(* PLC project Sin nombre, Desconocido Sin nombre 1 *)
(* stored: creationDateTime 2024-10-27T00:44:48, modificationDateTime 2024-10-28T16:29:27 *)

PROGRAM program0
  VAR
    timer : BOOL := 1;
    probar_sig : BOOL := 0;
    entro : BOOL := 0;
    entro0 : BOOL := 0;
    timer_corrido : BOOL := 0;
    acumular : BOOL := 0;
    hubo_cambio : BOOL := 0;  (* 0 *)
    luz1 : BOOL := 0;  (* darle ubic *)
    luz2 : BOOL := 0;  (* darle ubic *)
  END_VAR
  VAR
    sensor AT %IW0.0 : UINT := 34500;
  END_VAR
  VAR
    acum : UINT := 60000;
    tope_normal : UINT := 60;
    tope_alto : UINT := 40000;
    tope_superior : UINT := 0;
    actual : INT := 3;
    TON2 : TON;
    TP0 : TP;
    TOF1 : TOF;
    TP3 : TP;
    TON1 : TON;
    TON4 : TON;
    TON3 : TON;
    TON0 : TON;
    TON6 : TON;
  END_VAR
  VAR  (* added by the conversion: wires and edge detectors of the diagram *)
    _ADD78_ENO : BOOL;
    _ADD78_OUT : UINT;
    _EQ5_ENO : BOOL;
    _EQ5_OUT : BOOL;
    _GE83_ENO : BOOL;
    _GE83_OUT : BOOL;
    _ADD16_ENO : BOOL;
    _ADD16_OUT : INT;
    _EQ32_ENO : BOOL;
    _EQ32_OUT : BOOL;
    _GE55_ENO : BOOL;
    _GE55_OUT : BOOL;
    _LT97_ENO : BOOL;
    _LT97_OUT : BOOL;
  END_VAR

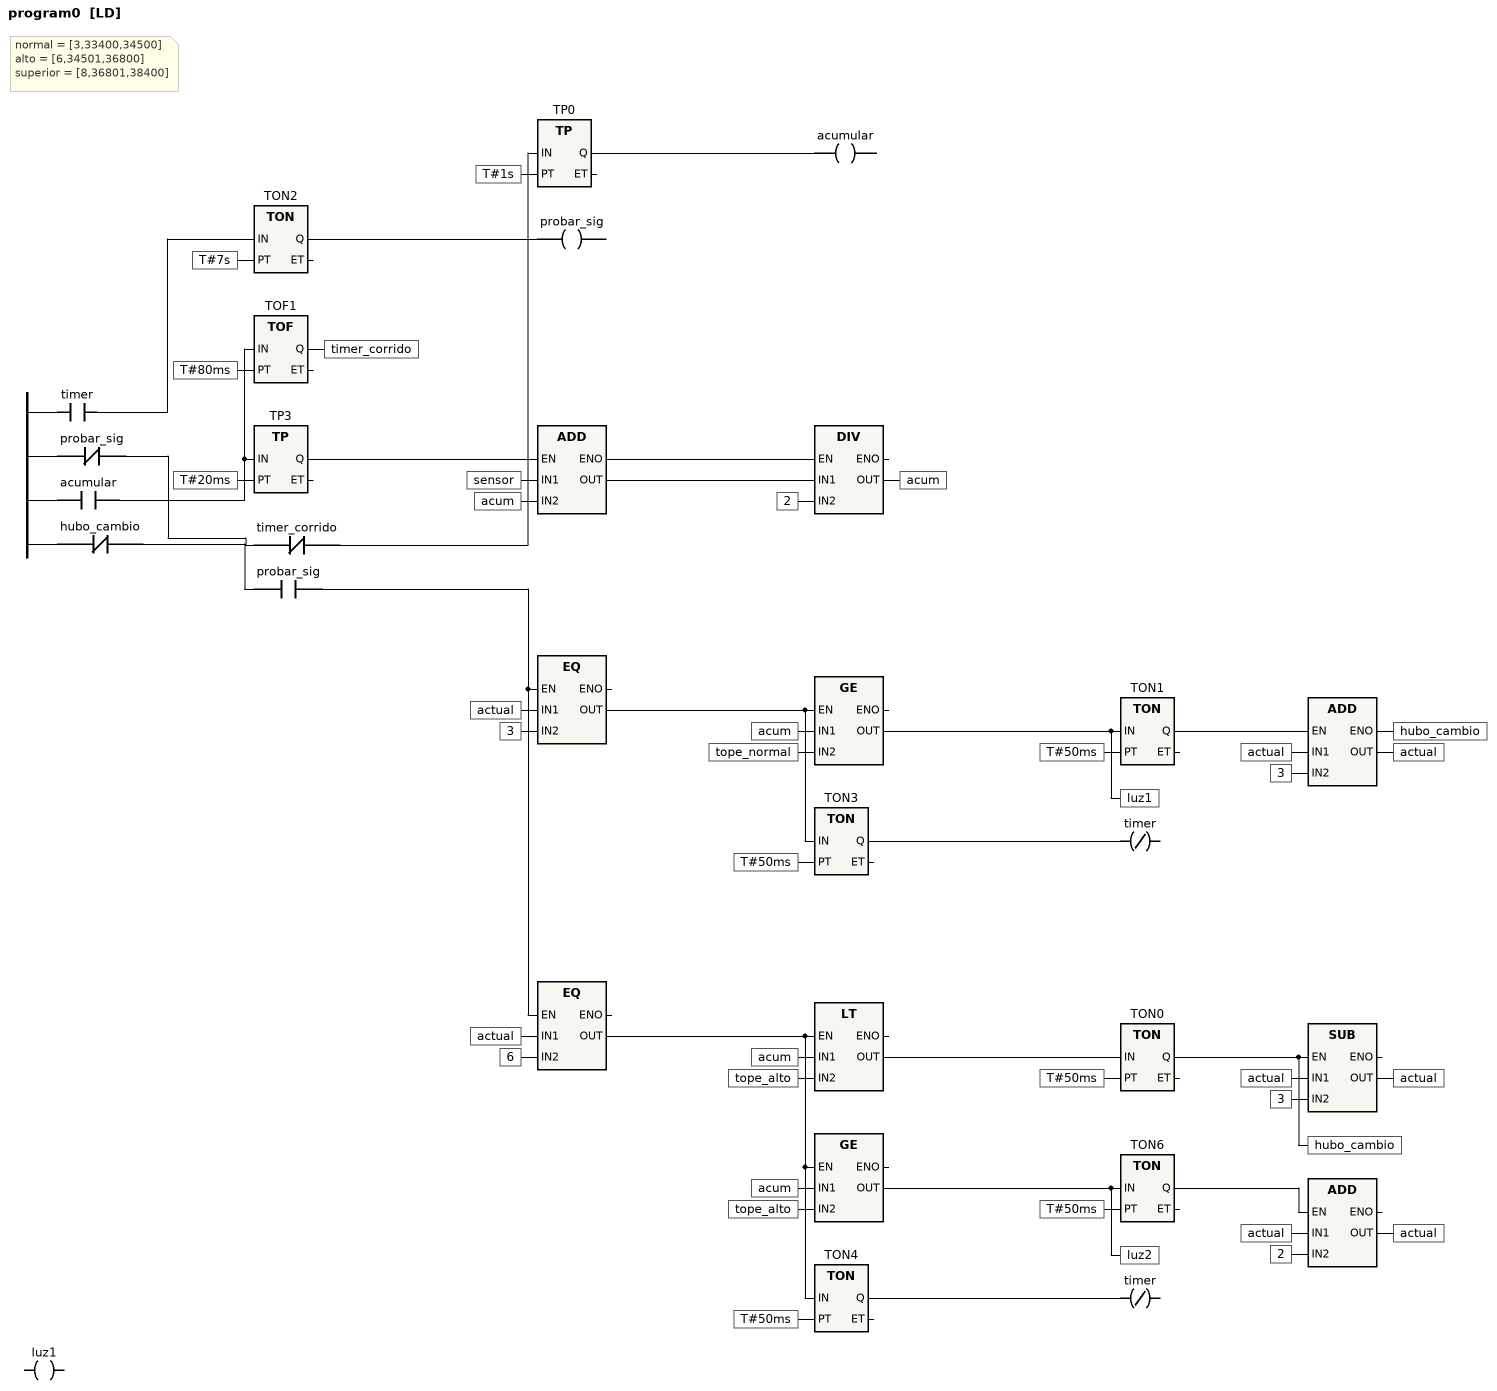
(* LD diagram, written out as Structured Text *)
TON2(IN := timer, PT := T#7s);
probar_sig := TON2.Q;
TP0(IN := NOT probar_sig AND NOT timer_corrido, PT := T#1s);
acumular := TP0.Q;
TOF1(IN := acumular, PT := T#80ms);
timer_corrido := TOF1.Q;
TP3(IN := acumular, PT := T#20ms);
_ADD78_OUT := ADD(EN := TP3.Q, IN1 := sensor, IN2 := acum, ENO => _ADD78_ENO);
IF _ADD78_ENO THEN acum := _ADD78_OUT / 2; END_IF;
(* normal = [3,33400,34500] 
    alto = [6,34501,36800]
    superior = [8,36801,38400] *)
_EQ5_OUT := EQ(EN := NOT hubo_cambio AND probar_sig, IN1 := actual, IN2 := 3, ENO => _EQ5_ENO);
_GE83_OUT := GE(EN := _EQ5_OUT, IN1 := acum, IN2 := tope_normal, ENO => _GE83_ENO);
TON1(IN := _GE83_OUT, PT := T#50ms);
_ADD16_OUT := ADD(EN := TON1.Q, IN1 := actual, IN2 := 3, ENO => _ADD16_ENO);
IF _ADD16_ENO THEN actual := _ADD16_OUT; END_IF;
_EQ32_OUT := EQ(EN := NOT hubo_cambio AND probar_sig, IN1 := actual, IN2 := 6, ENO => _EQ32_ENO);
_GE55_OUT := GE(EN := _EQ32_OUT, IN1 := acum, IN2 := tope_alto, ENO => _GE55_ENO);
TON6(IN := _GE55_OUT, PT := T#50ms);
IF TON6.Q THEN actual := actual + 2; END_IF;
_LT97_OUT := LT(EN := _EQ32_OUT, IN1 := acum, IN2 := tope_alto, ENO => _LT97_ENO);
TON0(IN := _LT97_OUT, PT := T#50ms);
IF TON0.Q THEN actual := actual - 3; END_IF;
TON4(IN := _EQ32_OUT, PT := T#50ms);
timer := NOT TON4.Q;
TON3(IN := _EQ5_OUT, PT := T#50ms);
timer := NOT TON3.Q;
IF _GE83_ENO THEN luz1 := _GE83_OUT; END_IF;
IF _GE55_ENO THEN luz2 := _GE55_OUT; END_IF;
hubo_cambio := TON0.Q;
hubo_cambio := _ADD16_ENO;
END_PROGRAM

CONFIGURATION Config0
  RESOURCE Res0 ON PLC
    TASK task0(INTERVAL := T#20ms, PRIORITY := 0);
    PROGRAM instance0 WITH task0 : program0;
  END_RESOURCE
END_CONFIGURATION
